INTERFACE I_ForcibleInt

{attribute 'monitoring' := 'call'}
PROPERTY Force : E_ForceState
GET
END_GET
SET
END_SET
END_PROPERTY

PROPERTY ForceValue : INT
GET
END_GET
SET
END_SET
END_PROPERTY

END_INTERFACE

(* stored: Version 1.1.0.1, ProductVersion 3.1.4026.18
   Itf I_ForcibleInt: Id {5cac6e74-4b9d-4f9c-8562-e709b70dd88d}
   Property Force: Id {8cbe7289-5ccd-4df2-b1d1-65ae1c15685f}
   Get Get: Id {33d20a49-af77-4ee9-a683-a66a914cc182}
   Set Set: Id {bb97807e-d5c8-4dfa-b10b-5a11e2f4cfdc}
   Property ForceValue: Id {aeaf6d33-87ea-4105-bab9-cb9c0d94cf49}
   Get Get: Id {8e83cb4f-29e8-4fa1-9c2e-2bfccd67960e}
   Set Set: Id {75be6d6d-1141-44cc-9e6a-34c37db14435} *)
